FUNCTION_BLOCK SEND_RECV_1_1 (* Send and receive on a duplex communication channel *)
  (* Standard: 61499-2; Description: Copyright (c) 2025 Martin Erich Jobst This program and the accompanying materials are made available under the terms of the Eclipse Public License 2.0 which is available at https://www.eclipse.org/legal/epl-2.0/ SPDX-License-Identifier: EPL-2.0 *)
  (* Version 3.0, 2025-07-11, Martin Erich Jobst, initial implementation *)
  PACKAGE iec61499::net;
  {SET_ATTRIBUTE(eclipse4diac::core::GenericClassName, 'GEN_SEND_RECV')}
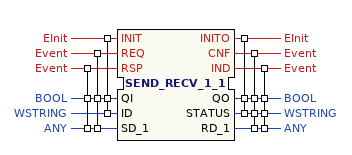
  EVENT_INPUT
    INIT : EInit WITH QI, ID; (* Service Initialization *)
    REQ WITH QI, SD_1; (* Send Request *)
    RSP WITH QI, SD_1; (* Receive Request *)
  END_EVENT
  EVENT_OUTPUT
    INITO : EInit WITH QO, STATUS; (* Initialization Confirm *)
    CNF WITH QO, STATUS, RD_1; (* Send Confirm *)
    IND WITH QO, STATUS, RD_1; (* Receive Indication *)
  END_EVENT
  VAR_INPUT
    QI : BOOL; (* Event Input Qualifier *)
    ID : WSTRING; (* Channel Identifier *)
    SD_1 : ANY; (* Data to Send *)
  END_VAR
  VAR_OUTPUT
    QO : BOOL; (* Event Output Qualifier *)
    STATUS : WSTRING; (* Channel Status *)
    RD_1 : ANY; (* Received Data *)
  END_VAR
END_FUNCTION_BLOCK
